
// ===== library: MasterCopy "WZAutomationLibDev" =====

VAR_GLOBAL   // PLC tag table "Tag table_1"
   "Sensor" AT %M100.0 : Bool;
   "DelayTime" AT %MD200 : Time;
   "DebounceMode" AT %MB102 : SInt;
   "TestStart" AT %M100.1 : Bool;
   "check" AT %M100.2 : Bool;
   "button" AT %M100.3 : Bool;
END_VAR

VAR_GLOBAL   // PLC tag table "Default tag table"
   "Clock_Byte" AT %MB0 : Byte;
   "Clock_10Hz" AT %M0.0 : Bool;
   "Clock_5Hz" AT %M0.1 : Bool;
   "Clock_2.5Hz" AT %M0.2 : Bool;
   "Clock_2Hz" AT %M0.3 : Bool;
   "Clock_1.25Hz" AT %M0.4 : Bool;
   "Clock_1Hz" AT %M0.5 : Bool;
   "Clock_0.625Hz" AT %M0.6 : Bool;
   "Clock_0.5Hz" AT %M0.7 : Bool;
   "System_Byte" AT %MB1 : Byte;
   "FirstScan" AT %M1.0 : Bool;
   "DiagStatusUpdate" AT %M1.1 : Bool;
   "AlwaysTRUE" AT %M1.2 : Bool;
   "AlwaysFALSE" AT %M1.3 : Bool;
END_VAR

DATA_BLOCK "WZALib_Debouncer_DB"   // DB1
{ S7_Optimized_Access := 'TRUE' }
AUTHOR : WZAutomation
VERSION : 0.1
// stored: InstanceOfName WZALib_Debouncer
"WZALib_Debouncer"
BEGIN
END_DATA_BLOCK

DATA_BLOCK "Block_1_DB"   // DB2
{ S7_Optimized_Access := 'TRUE' }
VERSION : 0.1
// stored: InstanceOfName Block_1
"Block_1"
BEGIN
END_DATA_BLOCK

DATA_BLOCK "WZALib_On/OffButton_DB"   // DB3
{ S7_Optimized_Access := 'TRUE' }
AUTHOR : WZAutomation
VERSION : 0.1
// stored: InstanceOfName WZALib_OnOffButton
"WZALib_OnOffButton"
BEGIN
END_DATA_BLOCK

FUNCTION_BLOCK "WZALib_Debouncer"   // FB1, SCL
TITLE = WZALib_Debouncer
{ S7_Optimized_Access := 'TRUE' }
AUTHOR : WZAutomation
VERSION : 0.1
// For more information, contact WZAutomation: contact@wzautomation.com. Use PLC system clock to perform time based boolean signal debounce hence the number of timer used for this purpose is significantly reduced.
   VAR_INPUT
      InSensor : Bool;   // Sensor to be debounced
      InDebounceTime : Time;   // Required debounce time in ms, max time = 10s
      InDebounceMode : SInt;   // Debounce mode, 0 = on/off debounce, 1 = on debounce, 2 = off debounce
   END_VAR
   VAR_OUTPUT
      OutSensorD : Bool;   // Sensor debounced
   END_VAR
   VAR
      Sensor_Mem : Bool;   // Sensor state from last PLC scan
      StateChangedto1R : R_TRIG;   // For On/Off debounce, rise edge of sensor state change 1st time
      SensorOnR : R_TRIG;   // For On debounce, rise edge when sensor turns on
      SensorOffR : R_TRIG;   // For Off debounce, rise edge when sensor turns off
      DebounceTime : Time;   // Actual debounce time according to input and check
      StateChange : CTU_SINT;
      PLC_SysTime : Date_And_Time;   // PLC local time read result
      "On/Off1stChange" : Date_And_Time := DT#2023-11-08-16:59:10;
      "On/OffDebounceTimeDiff" : Time;
      On1stChange : Date_And_Time;
      OnDebounceTimeDiff : Time;
      Off1stChange : Date_And_Time;
      OffDebounceTimeDiff : Time;
   END_VAR
   VAR_TEMP
      RD_SYS_T_Ret : Int;
   END_VAR
   VAR CONSTANT
      "On/Off" : SInt := 0;
      On : SInt := 1;
      Off : SInt := 2;
   END_VAR
BEGIN
   (*----------------------------------------------------------------------------------------------------------------------------------------------*
   *WZAutomationLib                                                                                                                                *
   *-----------------------------------------------------------------------------------------------------------------------------------------------*
   *Debounce mode 0: either sensor turns on or off will trigger a delay time defined by input and the sensor output is only changed if the input   *
   *sensor state is kept consistent during the time.                                                                                               *
   *Debounce mode 1: the debounce time is applied when sensor input is turned from off to on. When the sensor input is turned from on to off, the  *
   *output change applies instantly.                                                                                                               *
   *Debounce mode 2: the debounce time is applied when sensor input is turned from on to off. When the sensor input is turned from off to on, the  *
   *output change applies instantly.                                                                                                               *
   *-----------------------------------------------------------------------------------------------------------------------------------------------*
   *For more information, contact WZAutomation: contact@wzautomation.com                                                                           *
   *                                                                                                                                               *
   *-----------------------------------------------------------------------------------------------------------------------------------------------*)
   //Read PLC local time
   #RD_SYS_T_Ret := RD_SYS_T(#PLC_SysTime);

   //Debounce time check
   IF #InDebounceTime > T#10s THEN
       #DebounceTime := T#10s;
   ELSE
       #DebounceTime := #InDebounceTime;
   END_IF;

   CASE #InDebounceMode OF
       #"On/Off":
           //Detect sensor state change and count the edge
           #StateChange(CU := #InSensor <> #Sensor_Mem,
                        PV := 0);

           //Reset counter input tags to make sure the counter can catch change right after the current scan
           #StateChange.CU := #StateChange.R := FALSE;

           #StateChangedto1R(CLK := #StateChange.CV = 1);

           //Update sensor state mem
           #Sensor_Mem := #InSensor;

           CASE #StateChange.CV OF
               0:  //If no sensor state change is detected, send the sensor state straight through
                   #OutSensorD := #InSensor;

               1:  //If sensor state changed once, check if the sensor state is maintained during the debounce time
                   //Snapshot system time when state change counter becomes 1 then calculate how much time it has been sitting there
                   IF #StateChangedto1R.Q THEN
                       #"On/Off1stChange" := #PLC_SysTime;
                   ELSE
                       #"On/OffDebounceTimeDiff" := #PLC_SysTime - #"On/Off1stChange";
                   END_IF;

                   //Change output state if sensor state doesn't change anymore, otherwise, maintain output unchanged
                   IF #"On/OffDebounceTimeDiff" >= #DebounceTime AND #InSensor = #Sensor_Mem THEN
                       #OutSensorD := #InSensor;
                       #"On/OffDebounceTimeDiff" := T#0s;
                       #StateChange.CV := 0;
                   END_IF;

               2:  //If sensor state changed twice, debounce
                   #StateChange.CV := 0;
                   #"On/OffDebounceTimeDiff" := T#0s;
                   #StateChangedto1R.CLK := FALSE;

               ELSE  //Anything else, reset counter and do nothing
                   #StateChange.CV := 0;
                   #"On/OffDebounceTimeDiff" := T#0s;
                   #StateChangedto1R.CLK := FALSE;

           END_CASE;

       #On:
           #SensorOnR(CLK := #InSensor);

           //Snapshot system time when sensor turns on then calculate how much time it has been sitting there
           IF #SensorOnR.Q THEN
               #On1stChange := #PLC_SysTime;
           ELSIF #InSensor THEN
               #OnDebounceTimeDiff := #PLC_SysTime - #On1stChange;
               IF #OnDebounceTimeDiff >= #DebounceTime THEN
                   #OnDebounceTimeDiff := T#0s;
                   #OutSensorD := TRUE;
               END_IF;

               //Avoid debounce time difference overflow
               IF #OnDebounceTimeDiff > T#10s THEN
                   #OnDebounceTimeDiff := T#0s;
               END_IF;

           ELSE
               #OnDebounceTimeDiff := T#0s;
               #OutSensorD := FALSE;
           END_IF;

       #Off:
           #SensorOffR(CLK := NOT #InSensor);

           //Snapshot system time when sensor turns off then calculate how much time it has been sitting there
           IF #SensorOffR.Q THEN
               #Off1stChange := #PLC_SysTime;
           ELSIF NOT #InSensor THEN
               #OffDebounceTimeDiff := #PLC_SysTime - #Off1stChange;
               IF #OffDebounceTimeDiff >= #DebounceTime THEN
                   #OffDebounceTimeDiff := T#0s;
                   #OutSensorD := FALSE;
               END_IF;

               //Avoid debounce time difference overflow
               IF #OffDebounceTimeDiff > T#10s THEN
                   #OffDebounceTimeDiff := T#0s;
               END_IF;

           ELSE
               #OffDebounceTimeDiff := T#0s;
               #OutSensorD := TRUE;
           END_IF;

       ELSE  // Else, do nothing
           ;
   END_CASE;
END_FUNCTION_BLOCK

FUNCTION_BLOCK "Block_1"   // FB2, GRAPH_PLUS
{ S7_Optimized_Access := 'TRUE' }
VERSION : 0.1
   VAR_INPUT
      OFF_SQ : Bool := false;   // Turn sequence off
      INIT_SQ : Bool := false;   // Set sequence to initial state
      ACK_EF : Bool := false;   // Acknowledge all errors and faults
      S_PREV : Bool := false;   // Output previous step in parameter S_NO
      S_NEXT : Bool := false;   // Indicate next step in parameter S_NO
      SW_AUTO : Bool := false;   // Automatic mode
      SW_TAP : Bool := false;   // Semiautomatic/switch with transition
      SW_TOP : Bool := false;   // Semiautomatic/ignore transition
      SW_MAN : Bool := false;   // Manual mode
      S_SEL : Int := 0;   // Select step to be output to S_NO
      S_ON : Bool := false;   // Activate step indicated in S_NO
      S_OFF : Bool := false;   // Deactivate step indicated S_NO
      T_PUSH : Bool := false;   // Enable transition to switch in semi automatic mode
   END_VAR
   VAR_OUTPUT
      S_NO : Int := 0;   // Step number
      S_MORE : Bool := false;   // More steps are available and can be shown in S_NO
      S_ACTIVE : Bool := false;   // Step indicated in S_NO is active
      ERR_FLT : Bool := false;   // Interlock or supervision group error
      AUTO_ON : Bool := false;   // Automatic mode is active
      TAP_ON : Bool := false;   // Semiautomatic mode/step with transition enabled
      TOP_ON : Bool := false;   // Semiautomatic mode/ignore transition enabled
      MAN_ON : Bool := false;   // Manual mode is active
   END_VAR
   VAR
      HMI_INFO : Array[0..8] of UInt;
      IF_PAR : G7_IfParPlus_V6;
      RT_DATA : G7_RTDataPlus_V6;   // Internal data area
      Trans1 : G7_TransitionPlus_V6;   // Transition structure
      Trans3 : G7_TransitionPlus_V6;   // Transition structure
      Trans4 : G7_TransitionPlus_V6;   // Transition structure
      Trans5 : G7_TransitionPlus_V6;   // Transition structure
      Trans7 : G7_TransitionPlus_V6;   // Transition structure
      Trans8 : G7_TransitionPlus_V6;   // Transition structure
      Trans10 : G7_TransitionPlus_V6;   // Transition structure
      Trans11 : G7_TransitionPlus_V6;   // Transition structure
      "Wait to start" : G7_StepPlus_V6;   // Step structure
      "Set test signal" : G7_StepPlus_V6;   // Step structure
      "Reset test signal" : G7_StepPlus_V6;   // Step structure
      "Set test signal again" : G7_StepPlus_V6;   // Step structure
      "Reset test signal again" : G7_StepPlus_V6;   // Step structure
      "Set test signal for long time" : G7_StepPlus_V6;   // Step structure
      "Kill test signal for short time" : G7_StepPlus_V6;   // Step structure
      Step9 : G7_StepPlus_V6;   // Step structure
      SINI : Array[0..1] of USInt;
      LSTT : Array[0..7] of USInt;
      ATAJ : Array[0..7] of USInt;
      ATAB : Array[0..7] of USInt;
      PSTT : Array[0..7] of USInt;
      NSTT : Array[0..7] of USInt;
      ASSJ : Array[0..7] of USInt;
      ASSB : Array[0..7] of USInt;
      PTTS : Array[0..7] of USInt;
      NTTS : Array[0..7] of USInt;
      SW_SQTS : Array[0..7] of USInt;
      SWITCH : Array[0..0] of USInt;
      TVX : Array[0..1] of USInt;
      TTX : Array[0..1] of USInt;
      TSX : Array[0..1] of USInt;
      S00X : Array[0..1] of USInt;
      SOFFX : Array[0..1] of USInt;
      SONX : Array[0..1] of USInt;
      SAX : Array[0..1] of USInt;
      SERRX : Array[0..8] of USInt;
      SMX : Array[0..8] of USInt;
      S0X : Array[0..8] of USInt;
      S1X : Array[0..8] of USInt;
      IL_ALARM_INST : Diag_Alarm;
      SUP_ALARM_INST : Diag_Alarm;
      STEP_TIME_ALARM_INST : Diag_Alarm;
      IEC_TIMER_INST : IEC_TIMER;
      TRANSACTION_FLAG : Bool := false;
   END_VAR
   // SINI[0] := 2;
   // LSTT[0] := 255;
   // LSTT[1] := 255;
   // LSTT[2] := 255;
   // ATAJ[1] := 1;
   // ATAJ[2] := 2;
   // ATAJ[3] := 3;
   // ATAB[1] := 1;
   // ATAB[2] := 2;
   // ATAB[3] := 3;
   // PSTT[1] := 1;
   // PSTT[2] := 2;
   // PSTT[3] := 3;
   // NSTT[0] := 1;
   // NSTT[1] := 2;
   // NSTT[2] := 3;
   // ASSJ[1] := 1;
   // ASSJ[2] := 2;
   // ASSJ[3] := 3;
   // ASSB[1] := 1;
   // ASSB[2] := 2;
   // ASSB[3] := 3;
   // PTTS[0] := 255;
   // PTTS[2] := 1;
   // PTTS[3] := 2;
   // NTTS[1] := 1;
   // NTTS[2] := 2;
   // NTTS[3] := 3;
   // TVX[0] := 16#1;
   // TTX[0] := 16#1;
   // TSX[0] := 16#1;
   // S00X[0] := 16#1;
   // SOFFX[0] := 16#1;
   // SONX[0] := 16#1;
   // SAX[0] := 16#1;
   // SERRX[0] := 16#1;
   // SMX[0] := 16#1;
   // S0X[0] := 16#1;
   // S1X[0] := 16#1;
   // LSTT[3] := 255;
   // ATAJ[4] := 4;
   // ATAB[4] := 4;
   // PSTT[4] := 4;
   // NSTT[3] := 4;
   // ASSJ[4] := 4;
   // ASSB[4] := 4;
   // PTTS[4] := 3;
   // NTTS[4] := 4;
   // LSTT[4] := 255;
   // LSTT[5] := 255;
   // ATAJ[5] := 5;
   // ATAJ[6] := 6;
   // ATAB[5] := 5;
   // ATAB[6] := 6;
   // PSTT[5] := 5;
   // PSTT[6] := 6;
   // NSTT[4] := 5;
   // NSTT[5] := 6;
   // ASSJ[5] := 5;
   // ASSJ[6] := 6;
   // ASSB[5] := 5;
   // ASSB[6] := 6;
   // PTTS[5] := 4;
   // PTTS[6] := 5;
   // NTTS[5] := 5;
   // NTTS[6] := 6;
   // LSTT[6] := 255;
   // ATAJ[7] := 7;
   // ATAB[7] := 7;
   // PSTT[7] := 7;
   // NSTT[6] := 7;
   // ASSJ[7] := 7;
   // ASSB[7] := 7;
   // PTTS[7] := 6;
   // NTTS[7] := 7;
BEGIN
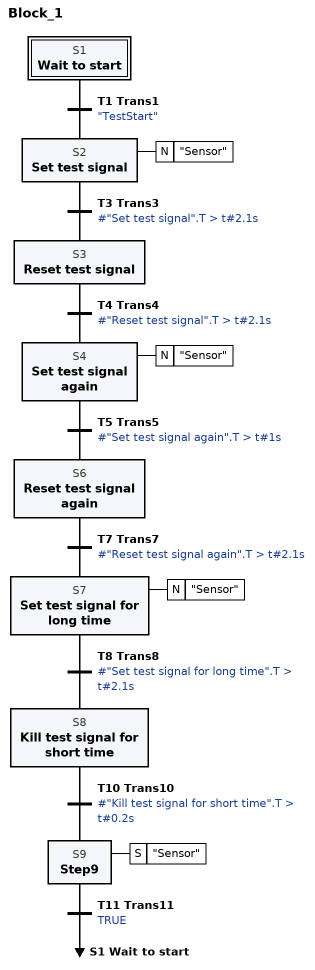
   // sequencer 1
   INITIAL_STEP "Wait to start":   // S1, max time T#10S, warning time T#7S
   END_STEP
   TRANSITION Trans1 FROM "Wait to start" TO "Set test signal"   // T1
      := "TestStart";
   END_TRANSITION
   STEP "Reset test signal":   // S3, max time T#10S, warning time T#7S
   END_STEP
   TRANSITION Trans4 FROM "Reset test signal" TO "Set test signal again"   // T4
      := #"Reset test signal".T > t#2.1s;
   END_TRANSITION
   STEP "Set test signal":   // S2, max time T#10S, warning time T#7S
              N    "Sensor"
   END_STEP
   TRANSITION Trans3 FROM "Set test signal" TO "Reset test signal"   // T3
      := #"Set test signal".T > t#2.1s;
   END_TRANSITION
   STEP "Set test signal again":   // S4, max time T#10S, warning time T#7S
              N    "Sensor"
   END_STEP
   TRANSITION Trans5 FROM "Set test signal again" TO "Reset test signal again"   // T5
      := #"Set test signal again".T > t#1s;
   END_TRANSITION
   STEP "Reset test signal again":   // S6, max time T#10S, warning time T#7S
   END_STEP
   TRANSITION Trans7 FROM "Reset test signal again" TO "Set test signal for long time"   // T7
      := #"Reset test signal again".T > t#2.1s;
   END_TRANSITION
   STEP "Set test signal for long time":   // S7, max time T#10S, warning time T#7S
              N    "Sensor"
   END_STEP
   TRANSITION Trans8 FROM "Set test signal for long time" TO "Kill test signal for short time"   // T8
      := #"Set test signal for long time".T > t#2.1s;
   END_TRANSITION
   STEP "Kill test signal for short time":   // S8, max time T#10S, warning time T#7S
   END_STEP
   TRANSITION Trans10 FROM "Kill test signal for short time" TO Step9   // T10
      := #"Kill test signal for short time".T > t#0.2s;
   END_TRANSITION
   STEP Step9:   // S9, max time T#10S, warning time T#7S
              S    "Sensor"
   END_STEP
   TRANSITION Trans11 FROM Step9 TO "Wait to start"   // T11, jump
      := TRUE;
   END_TRANSITION
END_FUNCTION_BLOCK

FUNCTION_BLOCK "WZALib_Sequencer"   // FB3, SCL
TITLE = WZALib_Sequencer
{ S7_Optimized_Access := 'TRUE' }
AUTHOR : WZAutomation
VERSION : 0.1
// For more information, contact WZAutomation: contact@wzautomation.com. Sequence control function block
   VAR_INPUT
      InAuto : Bool;   // Set sequence in auto mode (automatic step forward if conditions are fulfilled)
      InStepMode : Bool;   // Set sequence in step mode
      InStepCmd : Bool;
      InInterlock : Bool;
      InHoldStepTimer : Bool;
      InDefaultStepTime : Time;
   END_VAR
   VAR_OUTPUT
      OutSequenceTimeOut : Bool;
      OutCurrentStep : Int;
      OutCurrentStepTime : Time;
   END_VAR
   VAR
      Steps : Array[0..255] of Bool;   // Steps
      CurrentStep : Int;
      NextStep : Int;
      StepActiveTime : TON_TIME;
   END_VAR
BEGIN
   (*----------------------------------------------------------------------------------------------------------------------------------------------*
   *WZAutomationLib                                                                                                                                *
   *-----------------------------------------------------------------------------------------------------------------------------------------      *
   *For sequence control up to 256 steps.                                                                                                          *
   *In a typical machine automation application, it is normal to control a machine in step sequences. SFC is a good choice though the language     *
   *is heavy comparing with others and most of the scenarios SFC's functions are not fully utilized. WZAutomation made this sequencer with years   *
   *of experience in machine automation.                                                                                                           *
   InAuto: the sequence will run if this input is true.
   InStepMode: the sequence will run in step mode if InAuto is true.
   InStepCmd: the sequence will only move one step each time when the step's transition condition is fulfilled and this input sees a rising edge.
   InInterlock: 



   *-----------------------------------------------------------------------------------------------------------------------------------------      *
   *For more information, contact WZAutomation: contact@wzautomation.com                                                                           *
   *                                                                                                                                               *
   *-----------------------------------------------------------------------------------------------------------------------------------------------*)
END_FUNCTION_BLOCK

FUNCTION_BLOCK "WZALib_OnOffButton"   // FB4, SCL
TITLE = WZALib_On/OffButton
{ S7_Optimized_Access := 'TRUE' }
AUTHOR : WZAutomation
VERSION : 0.1
// For more information, contact WZAutomation: contact@wzautomation.com. For physical button to be pushed once to turn on and 2nd push to turn off.
   VAR_INPUT
      InButton : Bool;   // Push button input signal
   END_VAR
   VAR_OUTPUT
      OutSwitch : Bool;   // Push button on/off state
   END_VAR
   VAR
      ButtonState : Bool;   // Button state for FB calculation
      InputFTrig : F_TRIG;   // Detect the input button signals falling edge
   END_VAR
BEGIN
   (*----------------------------------------------------------------------------------------------------------------------------------------------*
   *WZAutomationLib                                                                                                                                *
   *-----------------------------------------------------------------------------------------------------------------------------------------------*
   *For single button input to alternate a boolean.                                                                                                *                                                                                          *
   *-----------------------------------------------------------------------------------------------------------------------------------------------*
   *For more information, contact WZAutomation: contact@wzautomation.com                                                                           *
   *                                                                                                                                               *
   *-----------------------------------------------------------------------------------------------------------------------------------------------*)

   //Catch the falling edge of the input button signal
   #InputFTrig(CLK := #InButton);

   //Generate button state based on memory
   IF #InputFTrig.Q AND #ButtonState THEN
       #ButtonState := FALSE;
   ELSIF #InputFTrig.Q AND NOT #ButtonState THEN
       #ButtonState := TRUE;
   END_IF;

   //Output the alternating state
   #OutSwitch := #ButtonState;
END_FUNCTION_BLOCK

ORGANIZATION_BLOCK "Main"   // OB1, LAD, ProgramCycle
TITLE = "Main Program Sweep (Cycle)"
{ S7_Optimized_Access := 'TRUE' }
VERSION : 0.1
   VAR_INPUT
      Initial_Call : Bool;   // Initial call of this OB
      Remanence : Bool;   // =True, if remanent data are available
   END_VAR
BEGIN

REGION Network 1
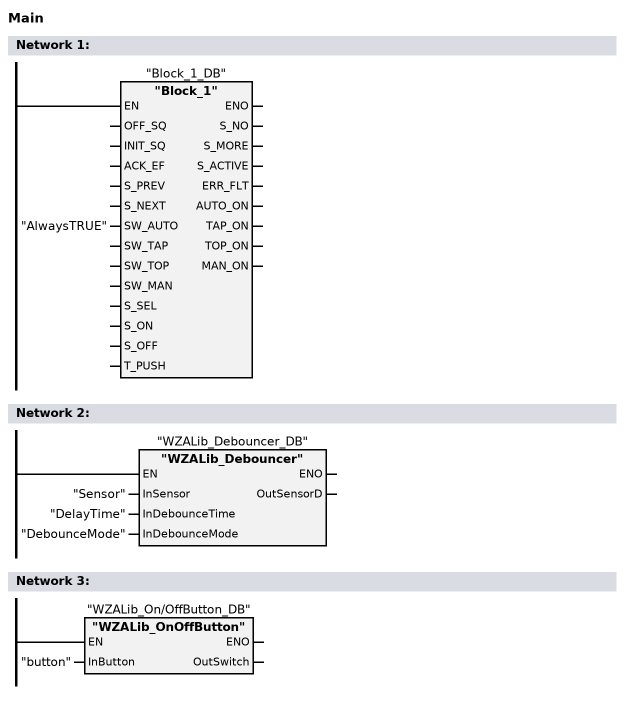
   RUNG wire#powerrail
      "Block_1_DB"(OFF_SQ :=, INIT_SQ :=, ACK_EF :=, S_PREV :=, S_NEXT :=, SW_AUTO := "AlwaysTRUE", SW_TAP :=, SW_TOP :=, SW_MAN :=, S_SEL :=, S_ON :=, S_OFF :=, T_PUSH :=, S_NO =>, S_MORE =>, S_ACTIVE =>, ERR_FLT =>, AUTO_ON =>, TAP_ON =>, TOP_ON =>, MAN_ON =>)
   END_RUNG
   // the same network as SCL:
   "Block_1_DB"(SW_AUTO := "AlwaysTRUE");   // "Block_1"
END_REGION

REGION Network 2
   RUNG wire#powerrail
      "WZALib_Debouncer_DB"(InSensor := "Sensor", InDebounceTime := "DelayTime", InDebounceMode := "DebounceMode", OutSensorD =>)
   END_RUNG
   // the same network as SCL:
   "WZALib_Debouncer_DB"(InSensor := "Sensor", InDebounceTime := "DelayTime", InDebounceMode := "DebounceMode");   // "WZALib_Debouncer"
END_REGION

REGION Network 3
   RUNG wire#powerrail
      "WZALib_On/OffButton_DB"(InButton := "button", OutSwitch =>)
   END_RUNG
   // the same network as SCL:
   "WZALib_On/OffButton_DB"(InButton := "button");   // "WZALib_OnOffButton"
END_REGION
END_ORGANIZATION_BLOCK

// ===== library: MasterCopy "PLC_1" =====

ORGANIZATION_BLOCK "Main"   // OB1, LAD, ProgramCycle
TITLE = "Main Program Sweep (Cycle)"
{ S7_Optimized_Access := 'TRUE' }
VERSION : 0.1
   VAR_INPUT
      Initial_Call : Bool;   // Initial call of this OB
      Remanence : Bool;   // =True, if remanent data are available
   END_VAR
BEGIN
END_ORGANIZATION_BLOCK